// TIA Portal V19 export
TYPE "LAF_typeConstraintRollerEm2ParametersInterface"
// stored: Access Published
   STRUCT
      configuration : "LAF_typeConstraintRollerEm2Parameters";
      commands : "LBC_typeInterfaceCommands";
      monitoring { S7_SetPoint := 'True'} : "LAF_typeConstraintRollerEm2ProcessValues";
   END_STRUCT;
END_TYPE
